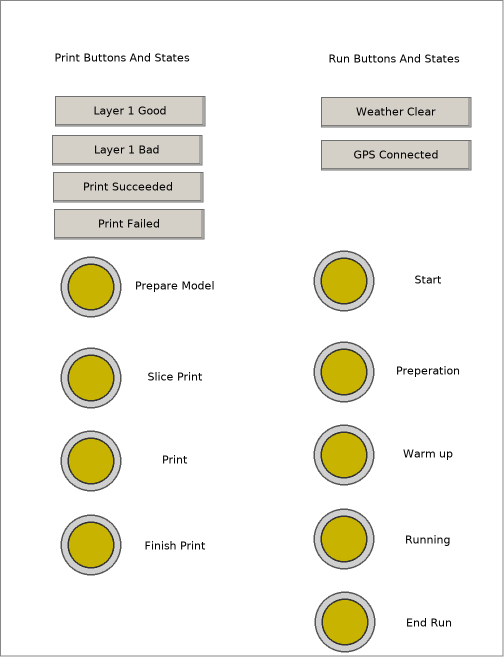
VISUALIZATION Visualization  // 504x657
    Button (321,97 150x30), "Weather Clear"
        tap Running2.WeatherClear
    Button (321,140 150x30), "GPS Connected"
        tap Running2.GPSConnected
    Button (55,96 150x30), "Layer 1 Good"
        tap GVL.Layer1Good
    Button (52,135 150x30), "Layer 1 Bad"
        tap GVL.Layer1Bad
    Lamp1 (56,252 70x70), variable: Printing.PrintStatePrepareModel, style: Lamp-Lamp1-Yellow
    Lamp1 (56,343 70x70), variable: Printing.PrintStateSlicePrint, style: Lamp-Lamp1-Yellow
    Lamp1 (56,426 70x70), variable: Printing.PrintStatePrint, style: Lamp-Lamp1-Yellow
    Lamp1 (56,510 70x70), variable: Printing.PrintStateFinishPrint, style: Lamp-Lamp1-Yellow
    Button (53,172 150x30), "Print Succeeded"
        tap Printing.PrintSucceeded
    Button (54,209 150x30), "Print Failed"
        tap GVL.Layer1Good
    Label (47,43 150x30), "Print Buttons And States"
    Label (100,271 150x30), "Prepare Model"
    Label (100,362 150x30), "Slice Print"
    Label (100,445 150x30), "Print"
    Label (100,531 150x30), "Finish Print"
    Label (319,44 150x30), "Run Buttons And States"
    Lamp1 (309,246 70x70), variable: Running2.RunstateStart, style: Lamp-Lamp1-Yellow
    Lamp1 (309,337 70x70), variable: Running2.RunstatePreperation, style: Lamp-Lamp1-Yellow
    Lamp1 (309,420 70x70), variable: Running2.RunstateWarmup, style: Lamp-Lamp1-Yellow
    Lamp1 (309,504 70x70), variable: Running2.RunstateRunning, style: Lamp-Lamp1-Yellow
    Label (353,265 150x30), "Start"
    Label (353,356 150x30), "Preperation"
    Label (353,439 150x30), "Warm up"
    Label (353,525 150x30), "Running"
    Lamp1 (310,587 70x70), variable: Running2.RunstateEndRun, style: Lamp-Lamp1-Yellow
    Label (354,608 150x30), "End Run"
END_VISUALIZATION

(* stored: Version 1.1.0.1, ProductVersion 3.1.4024.15
   Visu Visualization: Id {f6181437-23ad-43e1-a16e-df1a61571175} *)
